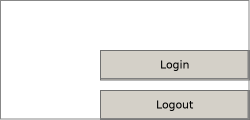
VISUALIZATION VISU_TEST_UserMgmt  // 250x120
    Button (100,50 150x30), "Login"
        OnMouseDown: VisuUserMgmt Type=Login
    Button (100,90 150x30), "Logout"
        OnMouseDown: VisuUserMgmt Type=Logout
END_VISUALIZATION

(* stored: Version 1.1.0.1, ProductVersion 3.1.4024.11
   Visu VISU_TEST_UserMgmt: Id {8eed0362-b648-0b1f-2601-52f470c11427} *)
